FUNCTION Convert_USINT_TO_TIME : Hresult
VAR_INPUT
	in : USINT;
	out : REFERENCE TO TIME;
END_VAR
VAR
	converted : TIME;
END_VAR

converted := USINT_TO_TIME(in);

IF (TIME_TO_USINT(converted) <> in) THEN
	Convert_USINT_TO_TIME := INCOMPATIBLE;
	RETURN;
END_IF

out := converted;

END_FUNCTION

(* stored: Version 1.1.0.1, ProductVersion 3.1.4024.12
   POU Convert_USINT_TO_TIME: Id {23519de0-6312-45b1-b2e7-2fe85ae56469}, SpecialFunc None *)
